GLOBALCONSTANTS DefaultPool_Horse_Numeric (* Numeric object pool constants (ID, Scale, Offset, Decimals) *)
  PACKAGE Uebungen::const::UT::Horse;
END_GLOBALCONSTANTS
